{attribute 'qualified_only'}
VAR_GLOBAL
	C1112_VTD_CIRCUIT_BREAKER AT%I*:BOOL;
	

END_VAR

(* stored: Version 1.1.0.1
   GVL IO_Panel: Id {1ae707b7-bb9a-4cd2-af2c-0476b860e240} *)
